# EPICS autosave request: iocBoot/iocARAmp/auto_settings_ARAmp50W1000DM2.req
file "aramp_settings_50W1000DM2.req",                P=$(P),  R=$(R)
